FUNCTION_BLOCK ADP_REPLAY100 (* Offline identification prototype; see docs/adaptive/4diac-design.md *)
  (* Standard: 61499-2 *)
  (* Version 0.1, 2026-09-26, Guilherme *)
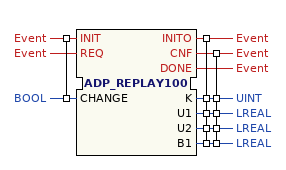
  EVENT_INPUT
    INIT WITH CHANGE;
    REQ;
  END_EVENT
  EVENT_OUTPUT
    INITO WITH K, U1, U2, B1;
    CNF WITH K, U1, U2, B1;
    DONE;
  END_EVENT
  VAR_INPUT
    CHANGE : BOOL := FALSE;
  END_VAR
  VAR_OUTPUT
    K : UINT;
    U1 : LREAL;
    U2 : LREAL;
    B1 : LREAL;
  END_VAR
  VAR
    NEXT_U : LREAL;
    CHANGE_ACTIVE : BOOL;
  END_VAR
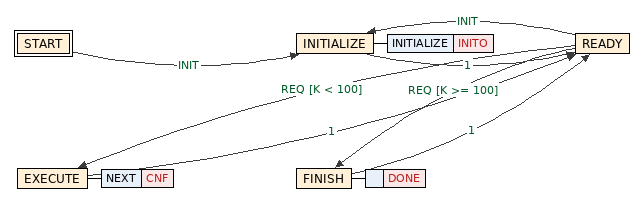
  EC_STATES
    START;
    INITIALIZE : INITIALIZE -> INITO;
    READY;
    EXECUTE : NEXT -> CNF;
    FINISH : -> DONE;
  END_STATES
  EC_TRANSITIONS
    START TO INITIALIZE := INIT;
    INITIALIZE TO READY := 1;
    READY TO INITIALIZE := INIT;
    READY TO EXECUTE := REQ [K < 100];
    READY TO FINISH := REQ [K >= 100];
    EXECUTE TO READY := 1;
    FINISH TO READY := 1;
  END_TRANSITIONS
  ALGORITHM INITIALIZE IN ST:
K := 0;
U1 := 0.0;
U2 := 0.0;
NEXT_U := 0.0;
B1 := 0.1;
CHANGE_ACTIVE := CHANGE;
  END_ALGORITHM
  ALGORITHM NEXT IN ST:
K := K + 1;
U2 := U1;
U1 := NEXT_U;
IF K = 1 THEN
NEXT_U := 0.0705087685450978;
END_IF;
IF K = 2 THEN
NEXT_U := 0.63490105216285753;
END_IF;
IF K = 3 THEN
NEXT_U := 0.080497931466046557;
END_IF;
IF K = 4 THEN
NEXT_U := 0.40763639883051483;
END_IF;
IF K = 5 THEN
NEXT_U := 0.61821610095614377;
END_IF;
IF K = 6 THEN
NEXT_U := 0.44427194683904436;
END_IF;
IF K = 7 THEN
NEXT_U := 0.8654313926360967;
END_IF;
IF K = 8 THEN
NEXT_U := 0.67760333389955507;
END_IF;
IF K = 9 THEN
NEXT_U := 0.12440745893021832;
END_IF;
IF K = 10 THEN
NEXT_U := 0.23061356841771596;
END_IF;
IF K = 11 THEN
NEXT_U := 0.34709955419584804;
END_IF;
IF K = 12 THEN
NEXT_U := 0.22692648606578547;
END_IF;
IF K = 13 THEN
NEXT_U := 0.019888601092231339;
END_IF;
IF K = 14 THEN
NEXT_U := 0.016162907429978057;
END_IF;
IF K = 15 THEN
NEXT_U := 0.73327763978997784;
END_IF;
IF K = 16 THEN
NEXT_U := 0.90228661094618257;
END_IF;
IF K = 17 THEN
NEXT_U := 0.19358927946656634;
END_IF;
IF K = 18 THEN
NEXT_U := 0.68232072221746187;
END_IF;
IF K = 19 THEN
NEXT_U := 0.54153806530301318;
END_IF;
IF K = 20 THEN
NEXT_U := 0.70649177482531711;
END_IF;
IF K = 21 THEN
NEXT_U := 0.30900800409617235;
END_IF;
IF K = 22 THEN
NEXT_U := 0.5244896510268896;
END_IF;
IF K = 23 THEN
NEXT_U := 0.15123674152649169;
END_IF;
IF K = 24 THEN
NEXT_U := 0.062828154370567435;
END_IF;
IF K = 25 THEN
NEXT_U := 0.11424592910182585;
END_IF;
IF K = 26 THEN
NEXT_U := 0.49673006525731844;
END_IF;
IF K = 27 THEN
NEXT_U := 0.041261524995094057;
END_IF;
IF K = 28 THEN
NEXT_U := 0.41058191707611214;
END_IF;
IF K = 29 THEN
NEXT_U := 0.15344703499761436;
END_IF;
IF K = 30 THEN
NEXT_U := 0.0089477299847484648;
END_IF;
IF K = 31 THEN
NEXT_U := 0.78546881976369309;
END_IF;
IF K = 32 THEN
NEXT_U := 0.77075549367531915;
END_IF;
IF K = 33 THEN
NEXT_U := 0.11488037289926367;
END_IF;
IF K = 34 THEN
NEXT_U := 0.81523353826384992;
END_IF;
IF K = 35 THEN
NEXT_U := 0.74778012039658015;
END_IF;
IF K = 36 THEN
NEXT_U := 0.22947350062996652;
END_IF;
IF K = 37 THEN
NEXT_U := 0.14582475407230944;
END_IF;
IF K = 38 THEN
NEXT_U := 0.56965077302758205;
END_IF;
IF K = 39 THEN
NEXT_U := 0.88996568691471034;
END_IF;
IF K = 40 THEN
NEXT_U := 0.8767654892239185;
END_IF;
IF K = 41 THEN
NEXT_U := 0.059518514937451306;
END_IF;
IF K = 42 THEN
NEXT_U := 0.34590115034707236;
END_IF;
IF K = 43 THEN
NEXT_U := 0.28913276235225682;
END_IF;
IF K = 44 THEN
NEXT_U := 0.27758989479536822;
END_IF;
IF K = 45 THEN
NEXT_U := 0.9334872688462611;
END_IF;
IF K = 46 THEN
NEXT_U := 0.93986591187291879;
END_IF;
IF K = 47 THEN
NEXT_U := 0.49261437515355266;
END_IF;
IF K = 48 THEN
NEXT_U := 0.82025863272654698;
END_IF;
IF K = 49 THEN
NEXT_U := 0.57370831231378638;
END_IF;
IF K = 50 THEN
NEXT_U := 0.32578329741873635;
END_IF;
IF K = 51 THEN
NEXT_U := 0.39438276329232402;
END_IF;
IF K = 52 THEN
NEXT_U := 0.4793713738430273;
END_IF;
IF K = 53 THEN
NEXT_U := 0.17003683157305782;
END_IF;
IF K = 54 THEN
NEXT_U := 0.79607914400863278;
END_IF;
IF K = 55 THEN
NEXT_U := 0.14453312469037671;
END_IF;
IF K = 56 THEN
NEXT_U := 0.45950688431666964;
END_IF;
IF K = 57 THEN
NEXT_U := 0.72150134876261018;
END_IF;
IF K = 58 THEN
NEXT_U := 0.36961795845763634;
END_IF;
IF K = 59 THEN
NEXT_U := 0.81086941727545081;
END_IF;
IF K = 60 THEN
NEXT_U := 0.33287739622808066;
END_IF;
IF K = 61 THEN
NEXT_U := 0.10755454143523469;
END_IF;
IF K = 62 THEN
NEXT_U := 0.73367887941811483;
END_IF;
IF K = 63 THEN
NEXT_U := 0.57705101697269612;
END_IF;
IF K = 64 THEN
NEXT_U := 0.72058160977576124;
END_IF;
IF K = 65 THEN
NEXT_U := 0.76897090955355607;
END_IF;
IF K = 66 THEN
NEXT_U := 0.32591725559758578;
END_IF;
IF K = 67 THEN
NEXT_U := 0.69114079455377242;
END_IF;
IF K = 68 THEN
NEXT_U := 0.10138596925555932;
END_IF;
IF K = 69 THEN
NEXT_U := 0.63115723249592448;
END_IF;
IF K = 70 THEN
NEXT_U := 0.56523729283117774;
END_IF;
IF K = 71 THEN
NEXT_U := 0.73792973304466358;
END_IF;
IF K = 72 THEN
NEXT_U := 0.42230559795399769;
END_IF;
IF K = 73 THEN
NEXT_U := 0.10355404067846252;
END_IF;
IF K = 74 THEN
NEXT_U := 0.24093230870479787;
END_IF;
IF K = 75 THEN
NEXT_U := 0.34135782007817272;
END_IF;
IF K = 76 THEN
NEXT_U := 0.65485529280356747;
END_IF;
IF K = 77 THEN
NEXT_U := 0.059810621354556393;
END_IF;
IF K = 78 THEN
NEXT_U := 0.52318569157328054;
END_IF;
IF K = 79 THEN
NEXT_U := 0.58992740962767998;
END_IF;
IF K = 80 THEN
NEXT_U := 0.74293679976989235;
END_IF;
IF K = 81 THEN
NEXT_U := 0.95692485111717762;
END_IF;
IF K = 82 THEN
NEXT_U := 0.95034473345133041;
END_IF;
IF K = 83 THEN
NEXT_U := 0.94641161661593465;
END_IF;
IF K = 84 THEN
NEXT_U := 0.65581835693723911;
END_IF;
IF K = 85 THEN
NEXT_U := 0.12966035605709103;
END_IF;
IF K = 86 THEN
NEXT_U := 0.36790878374028124;
END_IF;
IF K = 87 THEN
NEXT_U := 0.75598408947316298;
END_IF;
IF K = 88 THEN
NEXT_U := 0.28416878496193887;
END_IF;
IF K = 89 THEN
NEXT_U := 0.44011394653205682;
END_IF;
IF K = 90 THEN
NEXT_U := 0.18025876067922764;
END_IF;
IF K = 91 THEN
NEXT_U := 0.50940176540275917;
END_IF;
IF K = 92 THEN
NEXT_U := 0.47955931440237665;
END_IF;
IF K = 93 THEN
NEXT_U := 0.32053841902869451;
END_IF;
IF K = 94 THEN
NEXT_U := 0.2865850575270511;
END_IF;
IF K = 95 THEN
NEXT_U := 0.72903820599412372;
END_IF;
IF K = 96 THEN
NEXT_U := 0.68537736840209829;
END_IF;
IF K = 97 THEN
NEXT_U := 0.41927219450476338;
END_IF;
IF K = 98 THEN
NEXT_U := 0.84425722363228928;
END_IF;
IF K = 99 THEN
NEXT_U := 0.80733319489940969;
END_IF;
IF K = 100 THEN
NEXT_U := 0.97688866134232466;
END_IF;
B1 := 0.1;
IF CHANGE_ACTIVE AND (K >= 51) THEN
B1 := 0.4;
END_IF;
  END_ALGORITHM
END_FUNCTION_BLOCK
